PROGRAM MAIN
VAR
	Counter :INT := 0;
	ReadData: INT;
END_VAR

Counter := Counter + 1;
GVL_TcpExchange.uReadData_TcpExchangeTask := Counter;

END_PROGRAM

(* stored: Version 1.1.0.1, ProductVersion 3.1.4024.12
   POU MAIN: Id {9d4466c5-d30b-470f-b143-01ed8fac27be}, SpecialFunc None *)
